FUNCTION_BLOCK InfluxdbMeasurement IMPLEMENTS InterfaceSQLParameters
VAR_INPUT
END_VAR
VAR_OUTPUT
END_VAR
VAR
	_measurement_name :T_MaxString;
END_VAR

{warning 'add method implementation '}
METHOD add_column : BOOL
VAR_INPUT
	paramater	: Tc3_Database.ST_ExpParameter;
END_VAR
END_METHOD

{warning 'add property implementation'}
PROPERTY cbParameters : UDINT
GET
END_GET
END_PROPERTY

{warning 'add property implementation'}
PROPERTY column_num : UDINT
GET
END_GET
END_PROPERTY

{warning 'add property implementation'}
PROPERTY insert_query_string : Tc2_System.T_MaxString
GET
END_GET
END_PROPERTY

{warning 'add property implementation'}
PROPERTY pParameters : PVOID
GET
END_GET
END_PROPERTY

{warning 'add property implementation'}
PROPERTY table_name : Tc2_System.T_MaxString
GET
table_name := _measurement_name;
END_GET
SET
_measurement_name := table_name;
END_SET
END_PROPERTY

END_FUNCTION_BLOCK

(* stored: Version 1.1.0.1, ProductVersion 3.1.4024.12
   POU InfluxdbMeasurement: Id {c9f9009b-7df8-4bfb-a99e-e8b24991e013}, SpecialFunc None
   Method add_column: Id {0419eaef-2c5b-47fc-8e5d-3814335c2e9d}
   Property cbParameters: Id {bc4045ac-7c2d-4492-bd8e-2ff311e120ce}
   Get Get: Id {90370096-074c-4890-9887-ad28ceaccc33}
   Property column_num: Id {eca81d0f-25e9-489d-b626-e7661f1ef5b1}
   Get Get: Id {ac4d11d5-a034-4aa9-a103-99c2360fd558}
   Property insert_query_string: Id {cf42c815-52c3-41aa-9ccf-1faa8ceabf32}
   Get Get: Id {af55dbc7-3de4-4f51-ad95-f44d8e8f24e9}
   Property pParameters: Id {0c9c87ed-dce5-4cd8-babb-bf4559332553}
   Get Get: Id {ceb5108e-6b4b-42c5-910d-6bd42682b381}
   Property table_name: Id {1030ae34-ffa9-483a-a2c5-a2dcb663bec2}
   Get Get: Id {ddbc3561-694f-49ba-8d86-494e5c45f136}
   Set Set: Id {f3097ada-6e4b-4019-90c4-b24e93e32951} *)
